// TIA Portal project "SCL" (V14)

(* hardware
DEVICE "S7-1200 station_1"  S7-1200 Station
   slot 0: "Rack_0"  S7-1200 Rack  Rack  V1.0
   slot 1: "PLC_1"  CPU 1214C DC/DC/DC  6ES7 214-1AG40-0XB0  V4.2
*)

// ===== PLC "PLC_1"  CPU 1214C DC/DC/DC =====

VAR_GLOBAL   // PLC tag table "Default tag table"
   "StartPump" AT %Q0.0 : Bool;
   "StopPump" AT %Q0.1 : Bool;
   "LevelSensor" AT %IW0 : Int;   // 0-100
   "PumpStatus" AT %I2.0 : Bool;
   "MinLevel" AT %IW2 : Int;
   "MaxLevel" AT %IW4 : Int;
END_VAR

DATA_BLOCK "ControleBombas_DB"   // DB1
{ S7_Optimized_Access := 'TRUE' }
VERSION : 0.1
// stored: InstanceOfName ControleBombas
"ControleBombas"
BEGIN
END_DATA_BLOCK

FUNCTION_BLOCK "ControleBombas"   // FB1, SCL
{ S7_Optimized_Access := 'TRUE' }
VERSION : 0.1
   VAR_TEMP
      Temp_1 : Bool;
      StartPump : Bool;
      StopPump : Bool;
      LevelSensor : Int;   // 0-100
      PumpStatus : Bool;
   END_VAR
   VAR CONSTANT
      MinLevel : Int := 20;
      MaxLevel : Int := 80;
   END_VAR
BEGIN

   // Controle de bombas
   //IF #StartPump AND (#LevelSensor >= #MinLevel) THEN
   //#PumpStatus := TRUE;
   //END_IF
   IF #StartPump OR (#LevelSensor < #MinLevel) THEN
       #PumpStatus := TRUE;
   END_IF
   IF #StopPump THEN
       #PumpStatus := FALSE;
   END_IF
END_FUNCTION_BLOCK

FUNCTION "Controle de bombas" : Void   // FC1, SCL
{ S7_Optimized_Access := 'TRUE' }
VERSION : 0.1
   VAR_TEMP
      StartPump : Bool;
      StopPump : Bool;
      LevelSensor : Int;   // 0-100
      PumpStatus : Bool;
   END_VAR
   VAR CONSTANT
      MinLevel : Int := 20;
      MaxLevel : Int := 80;
   END_VAR
BEGIN

       // Controle de bombas
       //IF #StartPump AND (#LevelSensor >= #MinLevel) THEN
           //#PumpStatus := TRUE;
       //END_IF
       IF #StartPump OR (#LevelSensor < #MinLevel) THEN
           #PumpStatus := TRUE;
       END_IF
       IF #StopPump THEN
           #PumpStatus := FALSE;
       END_IF
END_FUNCTION

ORGANIZATION_BLOCK "Main"   // OB1, LAD, ProgramCycle
TITLE = "Main Program Sweep (Cycle)"
{ S7_Optimized_Access := 'TRUE' }
VERSION : 0.1
   VAR_INPUT
      Initial_Call : Bool;   // Initial call of this OB
      Remanence : Bool;   // =True, if remanent data are available
   END_VAR
BEGIN

REGION Network 1
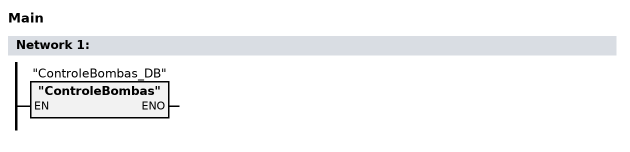
   RUNG wire#powerrail
      "ControleBombas_DB"()
   END_RUNG
   // the same network as SCL:
   "ControleBombas_DB"();   // "ControleBombas"
END_REGION
END_ORGANIZATION_BLOCK